// TIA Portal V16 export
// export: Created 2022-02-09T08:35:34.9317773Z, ExportSetting WithDefaults, DisplayName Totally Integrated Automation Portal, DisplayVersion V16 Update 5, DisplayName TIA Portal Version Control Interface, DisplayVersion V16 Update 2, DisplayName TIA Portal Openness, DisplayVersion V16 Update 5, DisplayName STEP 7 Professional, DisplayVersion V16 Update 5, DisplayName STEP 7 Safety, DisplayVersion V16, DisplayName WinCC Professional, DisplayVersion V16 Update 5, DisplayName SIMATIC Visualization Architect, DisplayVersion V16
FUNCTION_BLOCK "fbObjEV_Pantalo"   // FB9103, LAD
{ S7_Optimized_Access := 'TRUE' }
VERSION : 0.1
// stored: AutoNumber false, IsIECCheckEnabled false, IsRetainMemResEnabled false, MemoryReserve 0, SetENOAutomatically false, UDAEnableTagReadback false
   VAR_INPUT
      eDP1_DirCiclo3 : Bool := FALSE;
      eDP1_DirByPass23 : Bool;
      eDP2_DirCiclo2 : Bool;
      eDP2_DirCiclo1 : Bool := TRUE;
      eDirNumCicloAuto : Int;
      eForzaByPass : Bool;
      tAla_Posicio : Time := t#5s;
      psEnaAuto : Bool := TRUE;
      psEnaManual : Bool := FALSE;
      psAnuConMov : Bool;
      psResetAlarma : Bool;
      mFirstScan : Bool;
      clock : "clocks";
      bSysOk : Bool;
   END_VAR
   VAR_OUTPUT
      aEV1_DirByPass : Bool;
      aEV2_DirCiclo2 : Bool;
      be_DirCiclo1 : Bool;
      be_DirCiclo2 : Bool;
      be_DirCiclo3 : Bool;
      be_DirNumCiclo : Int;
      alDP1_DirCiclo1 : Bool := FALSE;
      alDP1_DirByPass : Bool;
      alDP2_DirCiclo2 : Bool;
      alDP2_DirCiclo3 : Bool := TRUE;
      iStatusDisplay : Int;
      bDisplayError : Bool;
      bDisplayWarning : Bool;
      bDisplayOk : Bool;
   END_VAR
   VAR
      psManDirByPass : Bool;
      psManDirCiclo2 : Bool;
      mDirNumCicloManual : Int;
      beDP1_DirCiclo1_Err : Bool := FALSE;
      beDP1_DirByPass_Err : Bool;
      beDP2_DirCiclo2_Err : Bool;
      beDP2_DirCiclo3_Err : Bool := TRUE;
      timAla_DirCiclo1 : IEC_TIMER;
      timAla_DirByPass : IEC_TIMER;
      timAla_DirCiclo2 { S7_SetPoint := 'True'} : IEC_TIMER;
      timAla_DirCiclo3 { S7_SetPoint := 'True'} : IEC_TIMER;
      mAuxTimer : Bool;
   END_VAR
   VAR_TEMP
      tmpNumCiclo : Int;
   END_VAR
   VAR CONSTANT
      STATUS_OBJ_ERR : Int := 10;
      STATUS_OBJ_WARNING : Int := 11;
      STATUS_OBJ_ON : Int := 1;
      STATUS_OBJ_OFF : Int := 0;
      STATUS_OBJ_UNKNOWN : Int := -1;
   END_VAR
   VAR_TEMP   // added for the SCL form of the ladder/FBD networks
      _w1 : Bool;
   END_VAR
BEGIN

REGION Network 1 (SCL): Descripció
   // Motor activat per Rele, amb confirmacio i proteccio.
END_REGION

REGION Network 2: Habilitació Mode Manual
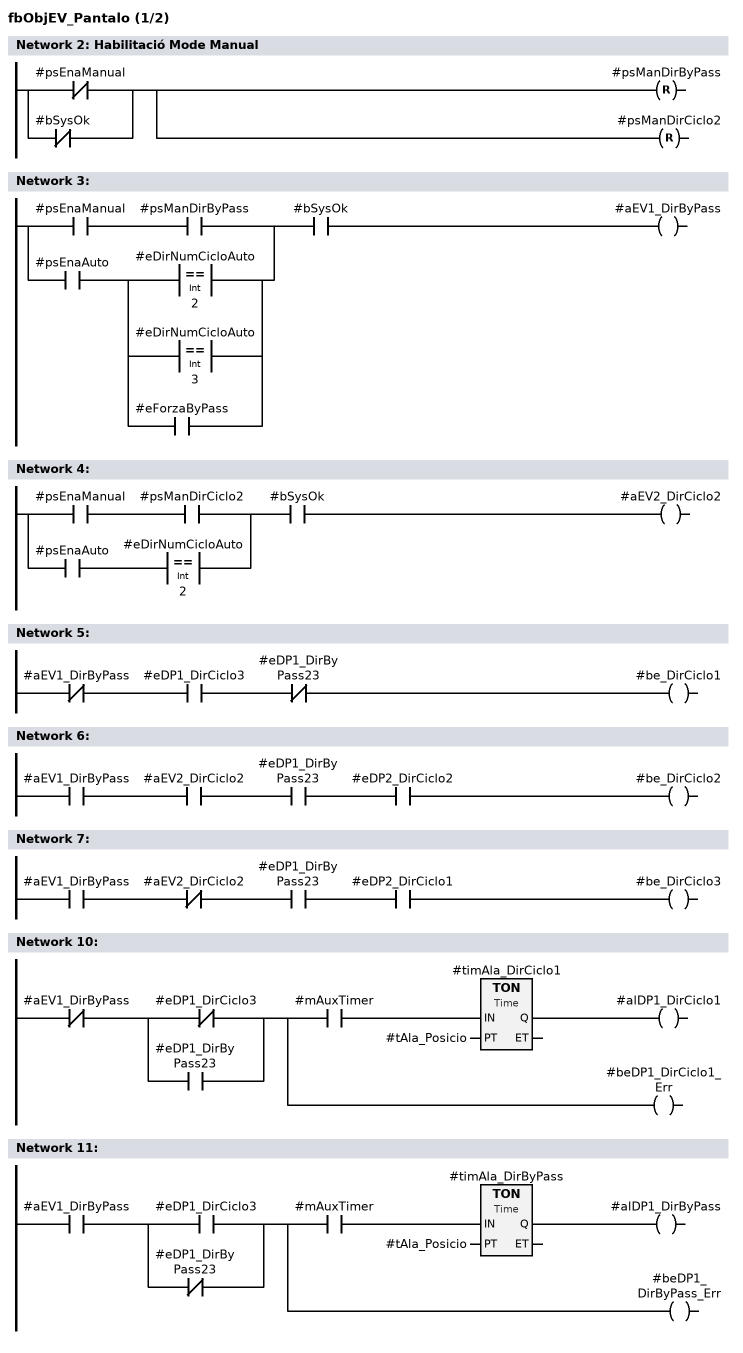
   RUNG wire#powerrail
      I_Contact( #psEnaManual )
      wire#w1
      R_Coil( #psManDirByPass )
   END_RUNG
   RUNG wire#powerrail
      I_Contact( #bSysOk )
   END_RUNG wire#w1
   RUNG wire#w1
      R_Coil( #psManDirCiclo2 )
   END_RUNG
   // the same network as SCL:
   IF NOT #psEnaManual OR NOT #bSysOk THEN
       #psManDirByPass := FALSE;
       #psManDirCiclo2 := FALSE;
   END_IF;
END_REGION

REGION Network 3
   RUNG wire#powerrail
      Contact( #psEnaManual )
      Contact( #psManDirByPass )
      wire#w1
      Contact( #bSysOk )
      Coil( #aEV1_DirByPass )
   END_RUNG
   RUNG wire#powerrail
      Contact( #psEnaAuto )
      wire#w2
      { S7_Templates := "SrcType := Int" } EQ_Contact(in1 := #eDirNumCicloAuto, in2 := 2)
   END_RUNG wire#w1
   RUNG wire#w2
      { S7_Templates := "SrcType := Int" } EQ_Contact(in1 := #eDirNumCicloAuto, in2 := 3)
   END_RUNG wire#w1
   RUNG wire#w2
      Contact( #eForzaByPass )
   END_RUNG wire#w1
   // the same network as SCL:
   #aEV1_DirByPass := ((#psEnaManual AND #psManDirByPass) OR (#psEnaAuto AND ((#eDirNumCicloAuto = 2) OR (#eDirNumCicloAuto = 3) OR #eForzaByPass))) AND #bSysOk;
END_REGION

REGION Network 4
   RUNG wire#powerrail
      Contact( #psEnaManual )
      Contact( #psManDirCiclo2 )
      wire#w1
      Contact( #bSysOk )
      Coil( #aEV2_DirCiclo2 )
   END_RUNG
   RUNG wire#powerrail
      Contact( #psEnaAuto )
      { S7_Templates := "SrcType := Int" } EQ_Contact(in1 := #eDirNumCicloAuto, in2 := 2)
   END_RUNG wire#w1
   // the same network as SCL:
   #aEV2_DirCiclo2 := ((#psEnaManual AND #psManDirCiclo2) OR (#psEnaAuto AND (#eDirNumCicloAuto = 2))) AND #bSysOk;
END_REGION

REGION Network 5
   RUNG wire#powerrail
      I_Contact( #aEV1_DirByPass )
      Contact( #eDP1_DirCiclo3 )
      I_Contact( #eDP1_DirByPass23 )
      Coil( #be_DirCiclo1 )
   END_RUNG
   // the same network as SCL:
   #be_DirCiclo1 := NOT #aEV1_DirByPass AND #eDP1_DirCiclo3 AND NOT #eDP1_DirByPass23;
END_REGION

REGION Network 6
   RUNG wire#powerrail
      Contact( #aEV1_DirByPass )
      Contact( #aEV2_DirCiclo2 )
      Contact( #eDP1_DirByPass23 )
      Contact( #eDP2_DirCiclo2 )
      Coil( #be_DirCiclo2 )
   END_RUNG
   // the same network as SCL:
   #be_DirCiclo2 := #aEV1_DirByPass AND #aEV2_DirCiclo2 AND #eDP1_DirByPass23 AND #eDP2_DirCiclo2;
END_REGION

REGION Network 7
   RUNG wire#powerrail
      Contact( #aEV1_DirByPass )
      I_Contact( #aEV2_DirCiclo2 )
      Contact( #eDP1_DirByPass23 )
      Contact( #eDP2_DirCiclo1 )
      Coil( #be_DirCiclo3 )
   END_RUNG
   // the same network as SCL:
   #be_DirCiclo3 := #aEV1_DirByPass AND NOT #aEV2_DirCiclo2 AND #eDP1_DirByPass23 AND #eDP2_DirCiclo1;
END_REGION

REGION Network 9 (SCL)
   IF #be_DirCiclo1 THEN
       #be_DirNumCiclo := 1;
   ELSIF #be_DirCiclo2 THEN
       #be_DirNumCiclo := 2;
   ELSIF #be_DirCiclo3 THEN
       #be_DirNumCiclo := 3;
   ELSE
       #be_DirNumCiclo := 0;
   END_IF;
END_REGION

REGION Network 10
   RUNG wire#powerrail
      I_Contact( #aEV1_DirByPass )
      wire#w1
      I_Contact( #eDP1_DirCiclo3 )
      wire#w2
      Contact( #mAuxTimer )
      { S7_Templates := "time_type := Time" } #timAla_DirCiclo1.TON(pt := #tAla_Posicio, et =>)
      Coil( #alDP1_DirCiclo1 )
   END_RUNG
   RUNG wire#w1
      Contact( #eDP1_DirByPass23 )
   END_RUNG wire#w2
   RUNG wire#w2
      Coil( #beDP1_DirCiclo1_Err )
   END_RUNG
   // the same network as SCL:
   #_w1 := NOT #aEV1_DirByPass AND (NOT #eDP1_DirCiclo3 OR #eDP1_DirByPass23);
   #timAla_DirCiclo1.TON(IN := #_w1 AND #mAuxTimer, PT := #tAla_Posicio);
   #alDP1_DirCiclo1 := #timAla_DirCiclo1.Q;
   #beDP1_DirCiclo1_Err := #_w1;
END_REGION

REGION Network 11
   RUNG wire#powerrail
      Contact( #aEV1_DirByPass )
      wire#w1
      Contact( #eDP1_DirCiclo3 )
      wire#w2
      Contact( #mAuxTimer )
      { S7_Templates := "time_type := Time" } #timAla_DirByPass.TON(pt := #tAla_Posicio, et =>)
      Coil( #alDP1_DirByPass )
   END_RUNG
   RUNG wire#w1
      I_Contact( #eDP1_DirByPass23 )
   END_RUNG wire#w2
   RUNG wire#w2
      Coil( #beDP1_DirByPass_Err )
   END_RUNG
   // the same network as SCL:
   #_w1 := #aEV1_DirByPass AND (#eDP1_DirCiclo3 OR NOT #eDP1_DirByPass23);
   #timAla_DirByPass.TON(IN := #_w1 AND #mAuxTimer, PT := #tAla_Posicio);
   #alDP1_DirByPass := #timAla_DirByPass.Q;
   #beDP1_DirByPass_Err := #_w1;
END_REGION

REGION Network 12
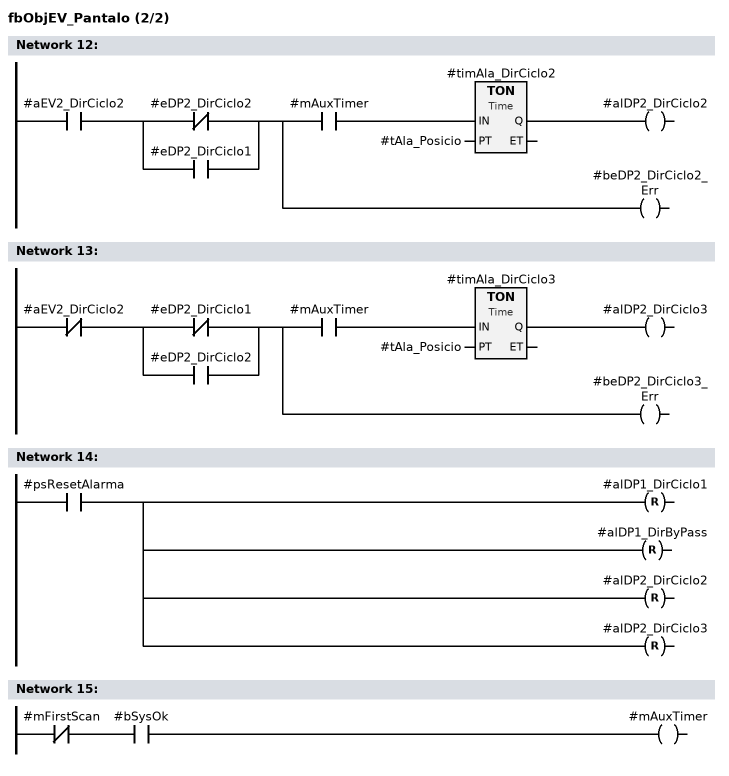
   RUNG wire#powerrail
      Contact( #aEV2_DirCiclo2 )
      wire#w1
      I_Contact( #eDP2_DirCiclo2 )
      wire#w2
      Contact( #mAuxTimer )
      { S7_Templates := "time_type := Time" } #timAla_DirCiclo2.TON(pt := #tAla_Posicio, et =>)
      Coil( #alDP2_DirCiclo2 )
   END_RUNG
   RUNG wire#w1
      Contact( #eDP2_DirCiclo1 )
   END_RUNG wire#w2
   RUNG wire#w2
      Coil( #beDP2_DirCiclo2_Err )
   END_RUNG
   // the same network as SCL:
   #_w1 := #aEV2_DirCiclo2 AND (NOT #eDP2_DirCiclo2 OR #eDP2_DirCiclo1);
   #timAla_DirCiclo2.TON(IN := #_w1 AND #mAuxTimer, PT := #tAla_Posicio);
   #alDP2_DirCiclo2 := #timAla_DirCiclo2.Q;
   #beDP2_DirCiclo2_Err := #_w1;
END_REGION

REGION Network 13
   RUNG wire#powerrail
      I_Contact( #aEV2_DirCiclo2 )
      wire#w1
      I_Contact( #eDP2_DirCiclo1 )
      wire#w2
      Contact( #mAuxTimer )
      { S7_Templates := "time_type := Time" } #timAla_DirCiclo3.TON(pt := #tAla_Posicio, et =>)
      Coil( #alDP2_DirCiclo3 )
   END_RUNG
   RUNG wire#w1
      Contact( #eDP2_DirCiclo2 )
   END_RUNG wire#w2
   RUNG wire#w2
      Coil( #beDP2_DirCiclo3_Err )
   END_RUNG
   // the same network as SCL:
   #_w1 := NOT #aEV2_DirCiclo2 AND (NOT #eDP2_DirCiclo1 OR #eDP2_DirCiclo2);
   #timAla_DirCiclo3.TON(IN := #_w1 AND #mAuxTimer, PT := #tAla_Posicio);
   #alDP2_DirCiclo3 := #timAla_DirCiclo3.Q;
   #beDP2_DirCiclo3_Err := #_w1;
END_REGION

REGION Network 14
   RUNG wire#powerrail
      Contact( #psResetAlarma )
      wire#w1
      R_Coil( #alDP1_DirCiclo1 )
   END_RUNG
   RUNG wire#w1
      R_Coil( #alDP1_DirByPass )
   END_RUNG
   RUNG wire#w1
      R_Coil( #alDP2_DirCiclo2 )
   END_RUNG
   RUNG wire#w1
      R_Coil( #alDP2_DirCiclo3 )
   END_RUNG
   // the same network as SCL:
   IF #psResetAlarma THEN
       #alDP1_DirCiclo1 := FALSE;
       #alDP1_DirByPass := FALSE;
       #alDP2_DirCiclo2 := FALSE;
       #alDP2_DirCiclo3 := FALSE;
   END_IF;
END_REGION

REGION Network 15
   RUNG wire#powerrail
      I_Contact( #mFirstScan )
      Contact( #bSysOk )
      Coil( #mAuxTimer )
   END_RUNG
   // the same network as SCL:
   #mAuxTimer := NOT #mFirstScan AND #bSysOk;
END_REGION

REGION Network 16 (SCL)
   IF #psEnaManual THEN
       IF (NOT #psManDirByPass) THEN
           #mDirNumCicloManual := 1;
       ELSIF (#psManDirCiclo2) THEN
           #mDirNumCicloManual := 2;
       ELSE
           #mDirNumCicloManual := 3;
       END_IF;
   ELSE
       #mDirNumCicloManual := 0;
       #tmpNumCiclo := #eDirNumCicloAuto;
   END_IF;

   // En cas de no tenir cap ciclo seleccionat, el valor en posicio de repos es Ciclo 1
   IF (#tmpNumCiclo = 0) THEN
       #tmpNumCiclo := 1;
   END_IF;
END_REGION

REGION Network 17 (SCL)
       IF (#alDP1_DirByPass OR #alDP1_DirCiclo1 OR #alDP2_DirCiclo2 OR #alDP2_DirCiclo3) THEN
           #iStatusDisplay := #STATUS_OBJ_ERR;                // Error = 10
           #bDisplayError := TRUE;
           #bDisplayWarning := FALSE;
           #bDisplayOk := FALSE;

       ELSIF (#beDP1_DirByPass_Err OR #beDP1_DirCiclo1_Err OR #beDP2_DirCiclo2_Err OR #beDP2_DirCiclo3_Err) THEN
           #iStatusDisplay := #STATUS_OBJ_WARNING;            // Warning = 11
           #bDisplayError := FALSE;
           #bDisplayWarning := TRUE;
           #bDisplayOk := FALSE;

       ELSIF #psEnaManual THEN
           // Hi ha activat mode manual. Pot ser que hi hagi sortides en auto o en manual.
           IF (#eDirNumCicloAuto > 0) THEN
               // Hi ha una seleccio en automatic. 
               IF (#eDirNumCicloAuto = #be_DirNumCiclo) THEN
                   // Si seleccio es la mateixa que en automatic (manual no modifica seleccio automatica)
                   #iStatusDisplay := #be_DirNumCiclo;
                   #bDisplayError := FALSE;
                   #bDisplayWarning := FALSE;
                   #bDisplayOk := TRUE;
               ELSE
                   // Si la seleccio difereix, indica que manual modifica la seleccio que fa el cicle automatic.
                   IF #clock."Clock_0.5Hz" THEN
                       #iStatusDisplay := #be_DirNumCiclo;
                       #bDisplayError := FALSE;
                       #bDisplayWarning := FALSE;
                       #bDisplayOk := TRUE;
                   ELSE
                       #iStatusDisplay := #be_DirNumCiclo;
                       #bDisplayError := FALSE;
                       #bDisplayWarning := TRUE;
                       #bDisplayOk := FALSE;
                   END_IF;
               END_IF;
           ELSE
               // No hi ha seleccio en automatic. Indiquem unicament els valors de seleccio en manual.
               #iStatusDisplay := #be_DirNumCiclo;
               #bDisplayError := FALSE;
               #bDisplayWarning := FALSE;
               #bDisplayOk := TRUE;
           END_IF;

       ELSIF (#eDirNumCicloAuto > 0) THEN
           // Posicionament en mode automatic
           IF (#eDirNumCicloAuto = #be_DirNumCiclo) THEN
               #iStatusDisplay := #be_DirNumCiclo;
               #bDisplayError := FALSE;
               #bDisplayWarning := FALSE;
               #bDisplayOk := TRUE;
           ELSE
               #iStatusDisplay := #STATUS_OBJ_WARNING;
               #bDisplayError := FALSE;
               #bDisplayWarning := TRUE;
               #bDisplayOk := FALSE;
           END_IF;

       ELSIF (#eDirNumCicloAuto = 0) THEN
           // No hi ha posicionament en mode automatic
           #iStatusDisplay := 1;
           #bDisplayError := FALSE;
           #bDisplayWarning := FALSE;
           #bDisplayOk := TRUE;

       ELSE
           #iStatusDisplay := #STATUS_OBJ_UNKNOWN;            // Unknown = -1
           #bDisplayError := TRUE;
           #bDisplayWarning := FALSE;
           #bDisplayOk := FALSE;

       END_IF;
END_REGION
END_FUNCTION_BLOCK
